// TIA Portal V17 export
// export: Created 2025-03-07T09:17:41.5944051Z, ExportSetting WithDefaults, DisplayName Totally Integrated Automation Portal, DisplayVersion V17 Update 8, DisplayName TIA Portal Openness, DisplayVersion V17 Update 8, DisplayName TIA Portal Version Control Interface, DisplayVersion V17, DisplayName SINAMICS Startdrive Advanced, DisplayVersion V17 SP2, DisplayName SINAMICS Startdrive G110M, G120, G120C, G120D, G120P, G115D, DisplayVersion V17 SP2, DisplayName SINAMICS Startdrive G130, G150, S120, S150, SINAMICS MV, S210, DisplayVersion V17 SP2, DisplayName STEP 7 Professional, DisplayVersion V17 Update 8, DisplayName SINUMERIK ONE STEP 7 Toolbox, DisplayVersion V17 Update 12, DisplayName SINUMERIK 840D sl STEP 7 Toolbox, DisplayVersion V17 Update 12, DisplayName STEP 7 Safety, DisplayVersion V17 Update 6, DisplayName WinCC Advanced, DisplayVersion V17 Update 8
FUNCTION "FC2002_BA_MODE" : Void   // FC2002, LAD
{ S7_Optimized_Access := 'FALSE' }
AUTHOR : ETXETAR
VERSION : 1.0
// stored: AutoNumber false, IsIECCheckEnabled false, SetENOAutomatically false, UDAEnableTagReadback false
   VAR_TEMP
      O_BYTE_0 : Struct   // OPTIONS BYTE 0
         BA_BUTTONS : Bool;   // BA MODE BUTTONS OPTION
         CHANGE_MODE_SEOC_ALARM : Bool;   // CHANGE MODE SEOC ALARM OPTION
         MODE_SELECTED_MEMORY : Bool;   // MODE SELECTED MEMORY OPTION
      END_STRUCT;
   END_VAR
   VAR CONSTANT
      FC_NUMBER : DInt := 2002;
   END_VAR
BEGIN

REGION Network 1: BA MODES MODE GROUP 1
   // 2#0000_0001 OPTIONS 0 BIT 0 BA BUTTONS
   // 2#0000_0010 OPTIONS 0 BIT 1 CHANGE MODE SEOC ALARM
   // 2#0000_0100 OPTIONS 0 BIT 2 MODE SELECTED MEMORY
   // 2#0000_1000 OPTIONS 0 BIT 3 SPARE
   // 2#0001_0000 OPTIONS 0 BIT 4 SPARE
   // 2#0010_0000 OPTIONS 0 BIT 5 SPARE
   // 2#0100_0000 OPTIONS 0 BIT 6 SPARE
   // 2#1000_0000 OPTIONS 0 BIT 7 SPARE
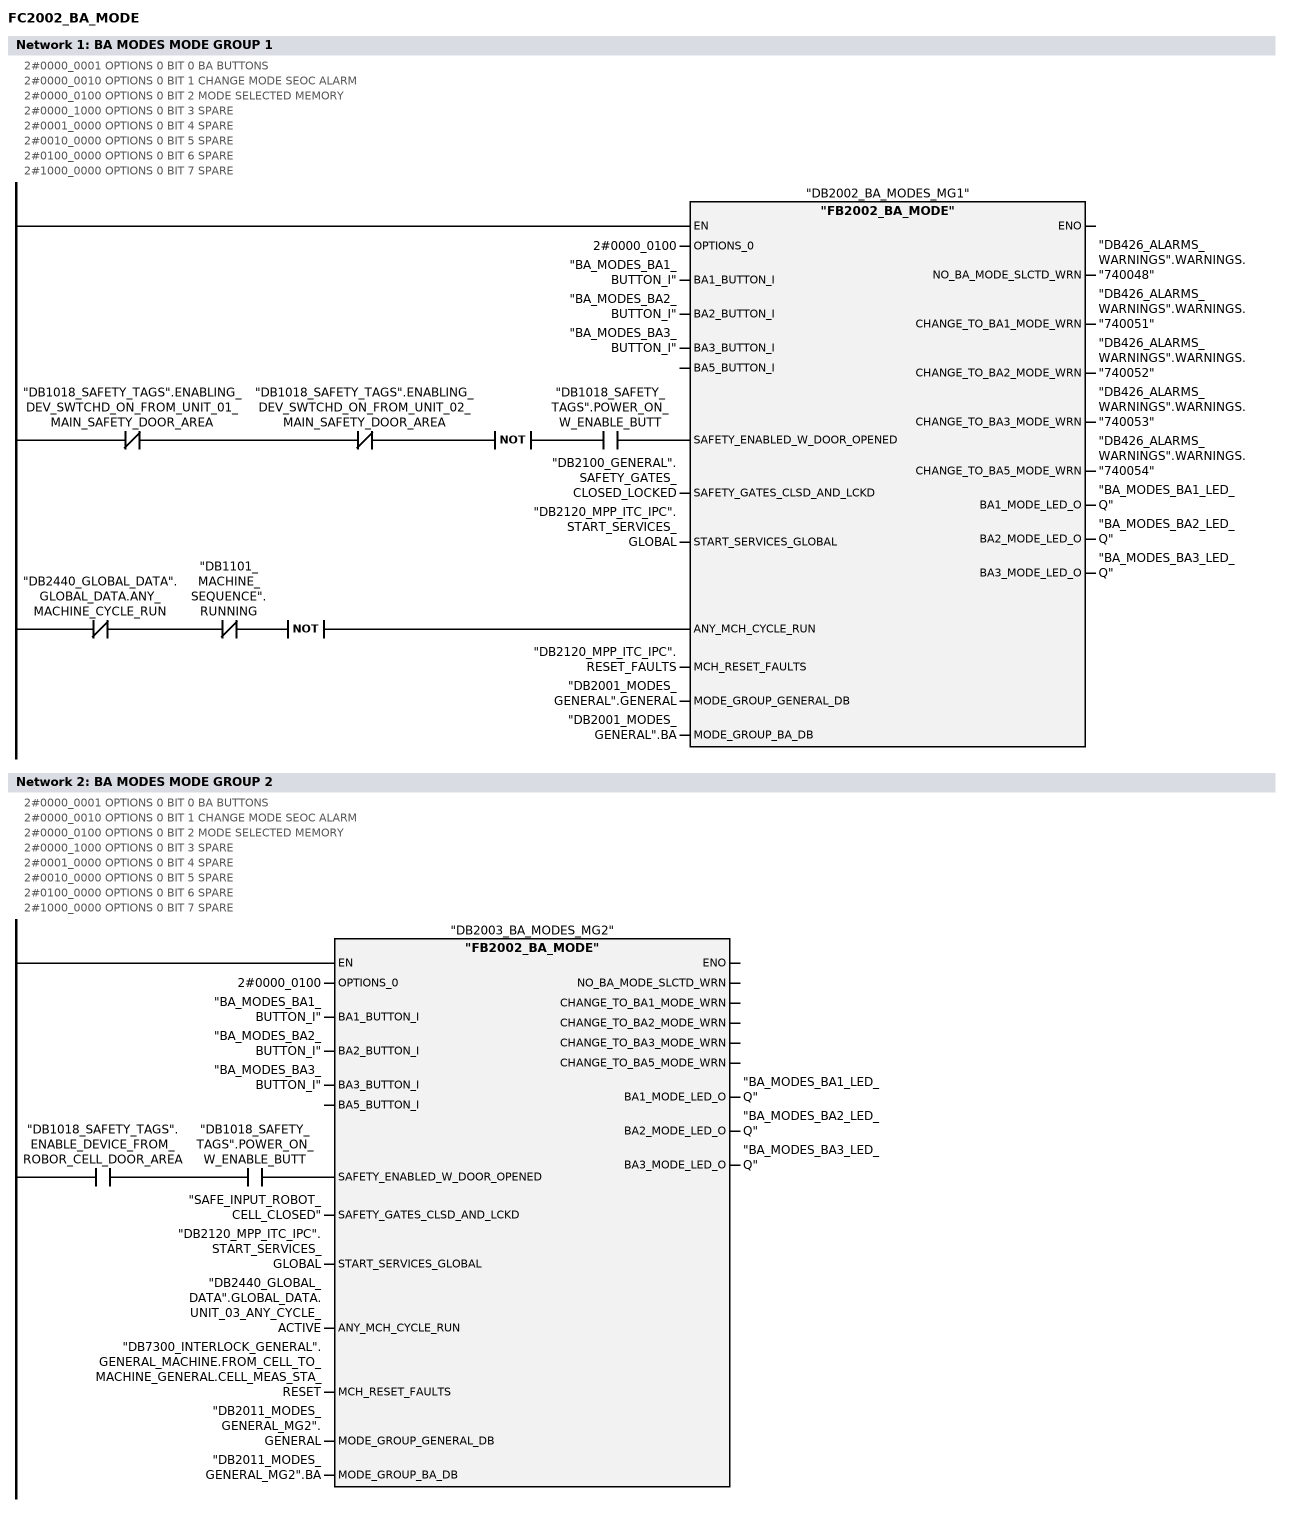
   RUNG wire#powerrail
      "DB2002_BA_MODES_MG1"(SAFETY_ENABLED_W_DOOR_OPENED := wire#w1, ANY_MCH_CYCLE_RUN := wire#w2, OPTIONS_0 := 2#0000_0100, BA1_BUTTON_I := "BA_MODES_BA1_BUTTON_I", BA2_BUTTON_I := "BA_MODES_BA2_BUTTON_I", BA3_BUTTON_I := "BA_MODES_BA3_BUTTON_I", BA5_BUTTON_I :=, SAFETY_GATES_CLSD_AND_LCKD := "DB2100_GENERAL".SAFETY_GATES_CLOSED_LOCKED, START_SERVICES_GLOBAL := "DB2120_MPP_ITC_IPC".START_SERVICES_GLOBAL, MCH_RESET_FAULTS := "DB2120_MPP_ITC_IPC".RESET_FAULTS, MODE_GROUP_GENERAL_DB := "DB2001_MODES_GENERAL".GENERAL, MODE_GROUP_BA_DB := "DB2001_MODES_GENERAL".BA, NO_BA_MODE_SLCTD_WRN => "DB426_ALARMS_WARNINGS".WARNINGS."740048", CHANGE_TO_BA1_MODE_WRN => "DB426_ALARMS_WARNINGS".WARNINGS."740051", CHANGE_TO_BA2_MODE_WRN => "DB426_ALARMS_WARNINGS".WARNINGS."740052", CHANGE_TO_BA3_MODE_WRN => "DB426_ALARMS_WARNINGS".WARNINGS."740053", CHANGE_TO_BA5_MODE_WRN => "DB426_ALARMS_WARNINGS".WARNINGS."740054", BA1_MODE_LED_O => "BA_MODES_BA1_LED_Q", BA2_MODE_LED_O => "BA_MODES_BA2_LED_Q", BA3_MODE_LED_O => "BA_MODES_BA3_LED_Q")
   END_RUNG
   RUNG wire#powerrail
      I_Contact( "DB1018_SAFETY_TAGS".ENABLING_DEV_SWTCHD_ON_FROM_UNIT_01_MAIN_SAFETY_DOOR_AREA )
      I_Contact( "DB1018_SAFETY_TAGS".ENABLING_DEV_SWTCHD_ON_FROM_UNIT_02_MAIN_SAFETY_DOOR_AREA )
      Not()
      Contact( "DB1018_SAFETY_TAGS".POWER_ON_W_ENABLE_BUTT )
   END_RUNG wire#w1
   RUNG wire#powerrail
      I_Contact( "DB2440_GLOBAL_DATA".GLOBAL_DATA.ANY_MACHINE_CYCLE_RUN )
      I_Contact( "DB1101_MACHINE_SEQUENCE".RUNNING )
      Not()
   END_RUNG wire#w2
   // the same network as SCL:
   "DB2002_BA_MODES_MG1"(OPTIONS_0 := 2#0000_0100,   // "FB2002_BA_MODE"
                         BA1_BUTTON_I := "BA_MODES_BA1_BUTTON_I",
                         BA2_BUTTON_I := "BA_MODES_BA2_BUTTON_I",
                         BA3_BUTTON_I := "BA_MODES_BA3_BUTTON_I",
                         SAFETY_ENABLED_W_DOOR_OPENED := NOT (NOT "DB1018_SAFETY_TAGS".ENABLING_DEV_SWTCHD_ON_FROM_UNIT_01_MAIN_SAFETY_DOOR_AREA AND NOT "DB1018_SAFETY_TAGS".ENABLING_DEV_SWTCHD_ON_FROM_UNIT_02_MAIN_SAFETY_DOOR_AREA) AND "DB1018_SAFETY_TAGS".POWER_ON_W_ENABLE_BUTT,
                         SAFETY_GATES_CLSD_AND_LCKD := "DB2100_GENERAL".SAFETY_GATES_CLOSED_LOCKED,
                         START_SERVICES_GLOBAL := "DB2120_MPP_ITC_IPC".START_SERVICES_GLOBAL,
                         ANY_MCH_CYCLE_RUN := NOT (NOT "DB2440_GLOBAL_DATA".GLOBAL_DATA.ANY_MACHINE_CYCLE_RUN AND NOT "DB1101_MACHINE_SEQUENCE".RUNNING),
                         MCH_RESET_FAULTS := "DB2120_MPP_ITC_IPC".RESET_FAULTS,
                         MODE_GROUP_GENERAL_DB := "DB2001_MODES_GENERAL".GENERAL,
                         MODE_GROUP_BA_DB := "DB2001_MODES_GENERAL".BA,
                         NO_BA_MODE_SLCTD_WRN => "DB426_ALARMS_WARNINGS".WARNINGS."740048",
                         CHANGE_TO_BA1_MODE_WRN => "DB426_ALARMS_WARNINGS".WARNINGS."740051",
                         CHANGE_TO_BA2_MODE_WRN => "DB426_ALARMS_WARNINGS".WARNINGS."740052",
                         CHANGE_TO_BA3_MODE_WRN => "DB426_ALARMS_WARNINGS".WARNINGS."740053",
                         CHANGE_TO_BA5_MODE_WRN => "DB426_ALARMS_WARNINGS".WARNINGS."740054",
                         BA1_MODE_LED_O => "BA_MODES_BA1_LED_Q",
                         BA2_MODE_LED_O => "BA_MODES_BA2_LED_Q",
                         BA3_MODE_LED_O => "BA_MODES_BA3_LED_Q");
END_REGION

REGION Network 2: BA MODES MODE GROUP 2
   // 2#0000_0001 OPTIONS 0 BIT 0 BA BUTTONS
   // 2#0000_0010 OPTIONS 0 BIT 1 CHANGE MODE SEOC ALARM
   // 2#0000_0100 OPTIONS 0 BIT 2 MODE SELECTED MEMORY
   // 2#0000_1000 OPTIONS 0 BIT 3 SPARE
   // 2#0001_0000 OPTIONS 0 BIT 4 SPARE
   // 2#0010_0000 OPTIONS 0 BIT 5 SPARE
   // 2#0100_0000 OPTIONS 0 BIT 6 SPARE
   // 2#1000_0000 OPTIONS 0 BIT 7 SPARE
   RUNG wire#powerrail
      "DB2003_BA_MODES_MG2"(SAFETY_ENABLED_W_DOOR_OPENED := wire#w1, OPTIONS_0 := 2#0000_0100, BA1_BUTTON_I := "BA_MODES_BA1_BUTTON_I", BA2_BUTTON_I := "BA_MODES_BA2_BUTTON_I", BA3_BUTTON_I := "BA_MODES_BA3_BUTTON_I", BA5_BUTTON_I :=, SAFETY_GATES_CLSD_AND_LCKD := "SAFE_INPUT_ROBOT_CELL_CLOSED", START_SERVICES_GLOBAL := "DB2120_MPP_ITC_IPC".START_SERVICES_GLOBAL, ANY_MCH_CYCLE_RUN := "DB2440_GLOBAL_DATA".GLOBAL_DATA.UNIT_03_ANY_CYCLE_ACTIVE, MCH_RESET_FAULTS := "DB7300_INTERLOCK_GENERAL".GENERAL_MACHINE.FROM_CELL_TO_MACHINE_GENERAL.CELL_MEAS_STA_RESET, MODE_GROUP_GENERAL_DB := "DB2011_MODES_GENERAL_MG2".GENERAL, MODE_GROUP_BA_DB := "DB2011_MODES_GENERAL_MG2".BA, NO_BA_MODE_SLCTD_WRN =>, CHANGE_TO_BA1_MODE_WRN =>, CHANGE_TO_BA2_MODE_WRN =>, CHANGE_TO_BA3_MODE_WRN =>, CHANGE_TO_BA5_MODE_WRN =>, BA1_MODE_LED_O => "BA_MODES_BA1_LED_Q", BA2_MODE_LED_O => "BA_MODES_BA2_LED_Q", BA3_MODE_LED_O => "BA_MODES_BA3_LED_Q")
   END_RUNG
   RUNG wire#powerrail
      Contact( "DB1018_SAFETY_TAGS".ENABLE_DEVICE_FROM_ROBOR_CELL_DOOR_AREA )
      Contact( "DB1018_SAFETY_TAGS".POWER_ON_W_ENABLE_BUTT )
   END_RUNG wire#w1
   // the same network as SCL:
   "DB2003_BA_MODES_MG2"(OPTIONS_0 := 2#0000_0100,   // "FB2002_BA_MODE"
                         BA1_BUTTON_I := "BA_MODES_BA1_BUTTON_I",
                         BA2_BUTTON_I := "BA_MODES_BA2_BUTTON_I",
                         BA3_BUTTON_I := "BA_MODES_BA3_BUTTON_I",
                         SAFETY_ENABLED_W_DOOR_OPENED := "DB1018_SAFETY_TAGS".ENABLE_DEVICE_FROM_ROBOR_CELL_DOOR_AREA AND "DB1018_SAFETY_TAGS".POWER_ON_W_ENABLE_BUTT,
                         SAFETY_GATES_CLSD_AND_LCKD := "SAFE_INPUT_ROBOT_CELL_CLOSED",
                         START_SERVICES_GLOBAL := "DB2120_MPP_ITC_IPC".START_SERVICES_GLOBAL,
                         ANY_MCH_CYCLE_RUN := "DB2440_GLOBAL_DATA".GLOBAL_DATA.UNIT_03_ANY_CYCLE_ACTIVE,
                         MCH_RESET_FAULTS := "DB7300_INTERLOCK_GENERAL".GENERAL_MACHINE.FROM_CELL_TO_MACHINE_GENERAL.CELL_MEAS_STA_RESET,
                         MODE_GROUP_GENERAL_DB := "DB2011_MODES_GENERAL_MG2".GENERAL,
                         MODE_GROUP_BA_DB := "DB2011_MODES_GENERAL_MG2".BA,
                         BA1_MODE_LED_O => "BA_MODES_BA1_LED_Q",
                         BA2_MODE_LED_O => "BA_MODES_BA2_LED_Q",
                         BA3_MODE_LED_O => "BA_MODES_BA3_LED_Q");
END_REGION
END_FUNCTION
